TYPE DUT_STRUCT_TEST :
STRUCT

	{attribute 'pytmc' := '
		pv: ADS_TST:fAmp
		io: o
		pv: ADS_TST:ReadOnly:fAmp
		io: i
	'}
	fAmplitude :	LREAL;
	{attribute 'pytmc' := '
		pv: ADS_TST:FArray
		io: o
		pv: ADS_TST:ReadOnly:FArray
		io: i
	'}
	fArray : ARRAY [1..5] OF LREAL;
	{attribute 'pytmc' := '
		pv: ADS_TST:Str
		io: o
		pv: ADS_TST:ReadOnly:Str
		io: i
	'}
	str	:	STRING(35);


END_STRUCT	
END_TYPE

(* stored: Version 1.1.0.1, ProductVersion 3.1.4022.18
   DUT DUT_STRUCT_TEST: Id {64b6492a-8751-410c-8dcd-b0346af5655e} *)
